// TwinCAT 3 PLC project MC2_Base
// ProgramVersion: 3.1.4024.0
// libraries:
//   Tc2_MC2, * (Beckhoff Automation GmbH)
//   Tc2_Standard, * (Beckhoff Automation GmbH)
//   Tc2_System, * (Beckhoff Automation GmbH)
//   Tc3_Module, * (Beckhoff Automation GmbH)
// project tree:
//   GVLs/ GVL.TcGVL (not stored)
//   / PlcTask.TcTTO
//   POUs/ FB_AxisBase.TcPOU, MAIN.TcPOU
// real-time tasks:
//   TASK PlcTask: cycle T#10ms, priority 20, ADS port 350
// motion (NC):
//   TASK NC-Task 1 SAF: cycle T#2ms, priority 4, ADS port 501
//   TASK NC-Task 1 SVB: cycle T#10ms, priority 8, ADS port 511
//   AXIS Achse 1 (id 1)
//     OtherSettings: AllowMotionCmdToSlave=true
//     encoder EncType=1
//     drive DrvType=5
//       Analog: TorqueSetpointScale=10, ScaleFactorActTorque=0.1
//     controller CtrType=1
//       CtrPara: PriorControlFactor=1
//         Observer: BandWidth=20
// variable links:
//   MC2_Base/MC2_Base Instance <-> NC-Task 1 SAF/Axes/Achse 1
//     PlcTask Inputs/GVL.axis_a.NcToPlc <-> Outputs/ToPlc
//     PlcTask Outputs/GVL.axis_a.PlcToNc <-> Inputs/FromPlc

CONFIGURATION MC2_Base
    RESOURCE PLC ON TwinCAT3
        TASK PlcTask(INTERVAL := T#10ms, PRIORITY := 20);
        PROGRAM MAIN WITH PlcTask : MAIN;
    END_RESOURCE
END_CONFIGURATION

// ---- POUs/MAIN.TcPOU
PROGRAM MAIN
VAR
	axis_a : FB_AxisBase := (	bStart	 		:= TRUE,
								bPowerEnable 	:= TRUE,
								bPosEnable 		:= TRUE,
								bNegEnable 		:= TRUE,
								fOverride 		:= 100.0);
								
	
END_VAR

axis_a(_axis_ref := GVL.axis_a);

END_PROGRAM

// ---- POUs/FB_AxisBase.TcPOU
FUNCTION_BLOCK FB_AxisBase
VAR_INPUT
	_axis_ref : REFERENCE TO AXIS_REF;
	
	bStart			: BOOL;
	bPowerEnable 	: BOOL;
	bPosEnable		: BOOL;
	bNegEnable		: BOOL;
	bStop			: BOOL;
	bReset 			: BOOL;
	fOverride		: LREAL := 0;
END_VAR
VAR_OUTPUT
	bAxisRdy		: BOOL;
	bError			: BOOL;
	nErrId			: UDINT;
END_VAR
VAR
	m_fb_power 	: MC_Power;
	m_fb_reset	: MC_Reset;
	m_fb_stop  	: MC_Stop;

	m_axis_status 	: ST_AxisStatus;
	m_state			: ST_McOutputs;
	st_fbMcStopOut	: ST_McOutputs;
	
	m_n_state		: UINT;
END_VAR

_axis_ref.ReadStatus();
m_axis_status := _axis_ref.Status;

IF bStart THEN
	bStart := FALSE;
	m_n_state := 10;
END_IF


CASE m_n_state OF
	0: // Idle	
		;

	10: // Enable Axis
		m_fb_power(
			Axis 				:= _axis_ref,
			Enable 				:= bPowerEnable,
			Override 			:= fOverride,
			Enable_Positive 	:= bPosEnable,
			Enable_Negative 	:= bNegEnable,
		);
		IF m_fb_power.Status THEN
			m_n_state := 20;
		END_IF
		
	20: // Axis Ready
		bAxisRdy := TRUE;
		m_n_state := 0;
	
END_CASE

	
m_fb_reset(
	Axis := _axis_ref,
	Execute := bReset
	);

	
m_fb_stop(
	Axis := _axis_ref,
	Execute := bStop,
	);


bStop 	:= FALSE;
bReset 	:= FALSE;

bError := m_fb_power.Error 		OR m_fb_reset.Error		OR m_fb_stop.Error;
nErrId := m_fb_power.ErrorID 	OR m_fb_reset.ErrorID	OR m_fb_stop.ErrorID;

END_FUNCTION_BLOCK
